FUNCTION_BLOCK E_TP (* standard timer function block (pulse) *)
  (* Standard: 61499-2; Classification: standard timer function block; Description: Copyright (c) 2024 HR Agrartechnik GmbH This program and the accompanying materials are made available under the terms of the Eclipse Public License 2.0 which is available at https://www.eclipse.org/legal/epl-2.0/ SPDX-License-Identifier: EPL-2.0 *)
  (* Version 3.1, 2026-05-13, Franz H??pfinger, HR Agrartechnik GmbH, E_R_TRIG instead of E_PERMIT *)
  (* Version 3.0, 2025-04-14, Patrick Aigner, changed package *)
  (* Version 1.1, 2024-04-23, Franz H??pfinger, HR Agrartechnik GmbH, Add a Reset to Timer FBs *)
  (* Version 1.0, 2024-03-04, Franz H??pfinger, HR Agrartechnik GmbH *)
  PACKAGE iec61499::events::timers;
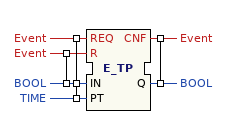
  EVENT_INPUT
    REQ WITH IN, PT; (* Service Request *)
    R WITH IN; (* Reset *)
  END_EVENT
  EVENT_OUTPUT
    CNF WITH Q; (* Confirmation of Requested Service *)
  END_EVENT
  VAR_INPUT
    IN : BOOL; (* Input *)
    PT : TIME; (* Pulse time *)
  END_VAR
  VAR_OUTPUT
    Q : BOOL; (* Output *)
  END_VAR
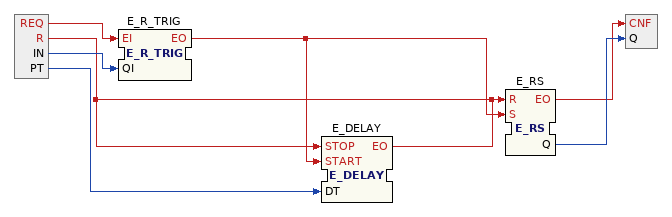
  FBS
    E_DELAY : iec61499::events::E_DELAY;
    E_RS : iec61499::events::E_RS;
    E_R_TRIG : iec61499::events::E_R_TRIG;
  END_FBS
  EVENT_CONNECTIONS
    E_RS.EO TO CNF;
    R TO E_DELAY.STOP;
    R TO E_RS.R;
    E_DELAY.EO TO E_RS.R;
    REQ TO E_R_TRIG.EI;
    E_R_TRIG.EO TO E_RS.S;
    E_R_TRIG.EO TO E_DELAY.START;
  END_CONNECTIONS
  DATA_CONNECTIONS
    PT TO E_DELAY.DT;
    E_RS.Q TO Q;
    IN TO E_R_TRIG.QI;
  END_CONNECTIONS
END_FUNCTION_BLOCK
